FUNCTION_BLOCK ResetTask EXTENDS TcoCore.TcoTask
VAR_IN_OUT
    rfidInOut : RfidInOut;
END_VAR
VAR_INPUT
    ActionDesc : STRING(25);
END_VAR
VAR
    _stringBuilder : TcoCore.StringBuilder;
    _state         : INT;

    _eErrorID   : RFID_FB_U.ERROR;
    _data       : Tc2_System.T_MaxString;
    _noTagFound : BOOL;

    _offSet : UDINT;

    _resetResponseCode : UINT := 16#8000;
END_VAR

IF (THIS^.Execute()) THEN

    CASE _state OF

        10:
            _state := 20;

        20:
            //Command setzen
            rfidInOut.eCommand := RFID_FB_U.COMMAND.RESET;
            _state             := 30;
        30:
            // Start der Operation
            rfidInOut.xExecute := TRUE;

            _state := 40;
        40:
            //            IF rfidInOut.stCompactModeInputMap.eResponseCode = _resetResponseCode THEN
            IF rfidInOut.xDone THEN
                THIS^.DoneWhen(TRUE);
                //                THIS^.Messenger.Info
                //                (
                //                    _stringbuilder.Append('Lock der Daten erfolgreich')
                //                        .Append('Startadresse: ')
                //                        .Append(TO_STRING(rfidinOut.udiStartAdress))
                //                        .Append(' Laenge: ')
                //                        .Append(TO_STRING(rfidInOut.uiDataLenght))
                //                        .ToString()
                //                );

                _state := 0;
            end_IF
    END_CASE
END_IF

{attribute 'monitoring' := 'call'}
PROPERTY ErrorId : RFID_FB_U.ERROR
GET
{warning disable C0371}
ErrorId := _eErrorID;
END_GET
END_PROPERTY

METHOD PUBLIC FB_init : BOOL
VAR_INPUT
    bInitRetains : BOOL; // if TRUE, the retain variables are initialized (warm start / cold start)
    bInCopyCode  : BOOL; // if TRUE, the instance afterwards gets moved into the copy code (online change)
    ParentObject : ITcoObject;
END_VAR
// This is not clear to me... I from time to time the consumer code does not see 'FB_init' of 'TcoObject', that's why overridden here with super call...
{warning disable C0316}
SUPER^.FB_init(bInitRetains, bInCopyCode, ParentObject);
END_METHOD

(*~
    <docu>
        <summary>
            Executes when task is aborted.
        </summary>
    </docu>
~*)
METHOD PROTECTED OnAbort
{warning disable C0371}
RfidInOut.eCommand := RFID_FB_U.COMMAND.IDLE;
RfidInOut.xExecute := FALSE;
RfidInOut.xAbort   := FALSE;
END_METHOD

(*~
    <docu>
        <summary>
            Executes when task reaches the ```Done``` state .
        </summary>
    </docu>
~*)
METHOD PROTECTED OnDone
{warning disable C0371}
rfidInOut.xExecute := FALSE;
rfidInOut.eCommand := RFID_FB_U.COMMAND.IDLE;
END_METHOD

(*~
    <docu>
        <summary>
            Executes when task reaches the ```Error``` state.
            <para>
                Do not confuse with <see cref="PlcDocu.TcoCore.TcoTask.WhileError()"/>, that is called cyclically until '''Error''' state is left.
            </para>
        </summary>
    </docu>
~*)
METHOD PROTECTED OnError
{warning disable C0371}
IF _noTagFound THEN
    _eErrorID := RFID_FB_U.ERROR.COMMAND_NO_TAG_FOUND;
    // not implemented by Turck
ELSIF rfidInOut.eErrorID = 16#2901 THEN
    _eErrorID := RFID_FB_U.ERROR.COMMAND_ADDRESS_OUTSIDE_BLOCK_BOUNDARIES;
ELSE
    _eErrorID := rfidInOut.eErrorID;
END_IF

THIS^.Messenger.Build().Append('Rfid Schreib/Lesekopf Fehler : ').Append(to_string(THIS^._eErrorID)).As().AsError();
END_METHOD

(*~
    <docu>
        <summary>
            Executes ones when the task starts (at the moment of transition from the ```Requested``` state into the ```Busy``` state).
        </summary>
    </docu>
~*)
METHOD PROTECTED OnStart
{warning disable C0371}
rfidInOut.eCommand := RFID_FB_U.COMMAND.IDLE;
rfidInOut.xExecute := FALSE;
rfidInOut.xAbort   := FALSE;
_state             := 10;
END_METHOD

(*~
    <docu>
        <summary>
            Restores this instance to the Ready state. Can be called explicitly or from within one of the restore mechanisms.
            <para>
                See also <see cref="PlcDocu.TcoCore.TcoTask.AutoRestorable()"/>
            </para>
        </summary>
    </docu>
~*)
METHOD Restore : ITcoRestorable
{warning disable C0371}
RfidInOut.eCommand := RFID_FB_U.COMMAND.IDLE;
RfidInOut.xExecute := FALSE;
RfidInOut.xAbort   := FALSE;
_noTagFound        := FALSE;
_eErrorID          := RFID_FB_U.ERROR.NO_ERROR;
SUPER^.Restore();
END_METHOD

END_FUNCTION_BLOCK

(* stored: Version 1.1.0.1, ProductVersion 3.1.4024.12
   POU ResetTask: Id {564eb7c5-50ae-097b-390c-a185cf54ec78}, SpecialFunc None
   Folder Status: Id {c15bae77-39e3-028c-22d8-86816e3ab073}
   Folder TcOpen: Id {61c131af-55f8-0bc1-154d-fe6b1d8aa9e0}
   Property ErrorId: Id {503ce27a-78e4-018b-14a5-1413e574e834}
   Get Get: Id {143ce37b-4840-0515-237f-61d296848cfd}
   Method FB_init: Id {6f970302-2417-0280-0fa1-5656c2c4253a}
   Method OnAbort: Id {25f60143-5596-01e1-3169-53ba83ddc52e}
   Method OnDone: Id {a5903579-2b31-0a1e-3e72-b78877903dab}
   Method OnError: Id {ea467b2e-1410-0925-357d-b1677a765e30}
   Method OnStart: Id {b3b7e549-1d61-09e4-1b77-65bebbb76663}
   Method Restore: Id {6cae50fe-33d8-08f7-2186-787f2dc693fe} *)
